// variable Geschwindigkeits Kontrolle
FUNCTION_BLOCK FB_SpeedControl
VAR_INPUT 
    viw_Speed : WORD; // Eingabe Soll-Geschwindigkeit
END_VAR
VAR_OUTPUT 
    vqx_VarSpeed : BOOL; // Enable Band Variable Geschwindigkeit
    vqw_Speed : WORD; // Band Soll-Geschwindigkeit
END_VAR
VAR 
    vsw_LastSpeed : WORD; // Soll-Geschwindigkeit von letztem Zyklus
	vtd_CalcSpeed: DINT;
	vtr_ScaleSpeed: REAL;
	vtr_NormSpeed: REAL;
END_VAR
VAR CONSTANT
	MAXNORM: INT := 27648;
	MINNORM: INT := 0;
	MAXSCALE: REAL := 100;
	MINSCALE: REAL := 0;
END_VAR

vqx_VarSpeed := TRUE;
IF (viw_Speed <> vsw_LastSpeed) THEN
    (*falls sich die Soll-Geschwindigkeit änderte*)
    (*Geschwindigkeit von WORD-Bereich auf Analogwert-Max skalieren*)   
	
 	vtd_CalcSpeed:= ABS(WORD_TO_DINT(viw_Speed)); //Wert in Absolutzahl speichern
	
	vtr_ScaleSpeed:= (MAXSCALE - MINSCALE)/ MAXNORM * DINT_TO_REAL(vtd_CalcSpeed) + MINSCALE;
	vtr_NormSpeed:= (((vtr_ScaleSpeed - MINSCALE) / (MAXSCALE - MINSCALE)) * (MAXNORM - MINNORM)) + MINNORM;
	vqw_Speed := INT_TO_WORD(REAL_TO_INT(vtr_NormSpeed));
    
	vsw_LastSpeed := viw_Speed; (*aktuelle Speed abspeichern für nächsten Zyklus*)
END_IF;

END_FUNCTION_BLOCK

(* stored: Version 1.1.0.1
   POU FB_SpeedControl: Id {00448bd9-e5a5-4404-8981-797a91c7cc5e}, SpecialFunc None *)
